// TwinCAT 3 PLC project CodeAnalysis
// ProgramVersion: 3.1.4022.3
// libraries:
//   Tc2_Standard, * (Beckhoff Automation GmbH)
//   Tc2_System, * (Beckhoff Automation GmbH)
//   Tc3_Module, * (Beckhoff Automation GmbH)
// project tree:
//   / PlcTask.TcTTO
//   POUs/ MAIN.TcPOU
// real-time tasks:
//   TASK PlcTask: cycle T#10ms, priority 20, ADS port 350

CONFIGURATION CodeAnalysis
    RESOURCE PLC ON TwinCAT3
        TASK PlcTask(INTERVAL := T#10ms, PRIORITY := 20);
        PROGRAM MAIN WITH PlcTask : MAIN;
    END_RESOURCE
END_CONFIGURATION

// ---- POUs/MAIN.TcPOU
PROGRAM MAIN
VAR
	bJustASimpleBoolean : BOOL; // SA0033 - WARNING
	sThisStringIsTooLong : STRING(6) := 'Hello world'; // SA0026 - ERROR
	
	nCounter : ULINT;
END_VAR

nCounter := nCounter + 1;

sThisStringIsTooLong := '';

END_PROGRAM
